// TIA Portal V19 export
FUNCTION "FC900_SafetyIntegration" : Void   // FC900, F_LAD
{ S7_Optimized_Access := 'TRUE' }
// stored: AutoNumber false
BEGIN

REGION Network 1: Bit de reset
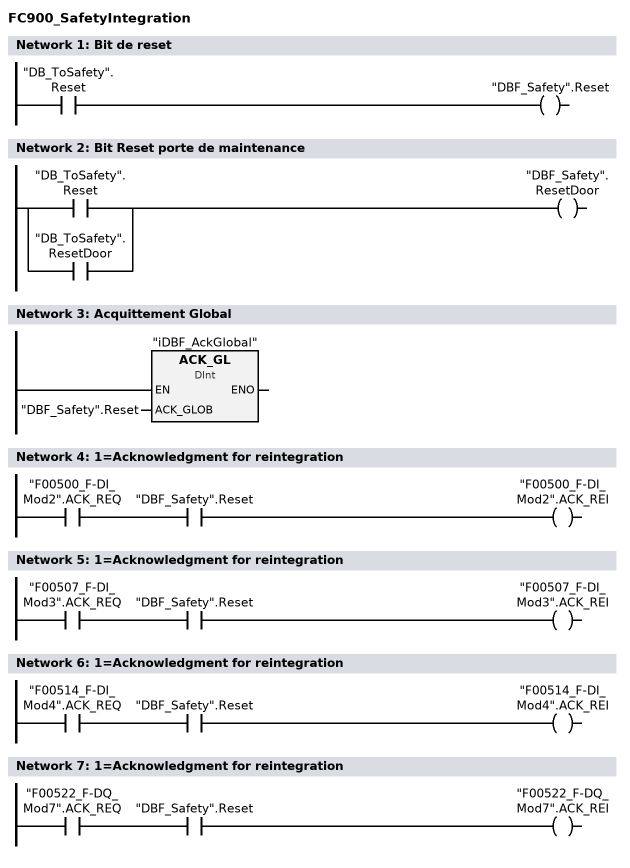
   RUNG wire#powerrail
      Contact( "DB_ToSafety".Reset )
      Coil( "DBF_Safety".Reset )
   END_RUNG
   // the same network as SCL:
   "DBF_Safety".Reset := "DB_ToSafety".Reset;
END_REGION

REGION Network 2: Bit Reset porte de maintenance
   RUNG wire#powerrail
      Contact( "DB_ToSafety".Reset )
      wire#w1
      Coil( "DBF_Safety".ResetDoor )
   END_RUNG
   RUNG wire#powerrail
      Contact( "DB_ToSafety".ResetDoor )
   END_RUNG wire#w1
   // the same network as SCL:
   "DBF_Safety".ResetDoor := "DB_ToSafety".Reset OR "DB_ToSafety".ResetDoor;
END_REGION

REGION Network 3: Acquittement Global
   RUNG wire#powerrail
      { S7_Templates := "codedbool_type := DInt" } "iDBF_AckGlobal".ACK_GL(ACK_GLOB := "DBF_Safety".Reset)
   END_RUNG
   // the same network as SCL:
   "iDBF_AckGlobal"(ACK_GLOB := "DBF_Safety".Reset);   // ACK_GL
END_REGION

REGION Network 4: 1=Acknowledgment for reintegration
   RUNG wire#powerrail
      Contact( "F00500_F-DI_Mod2".ACK_REQ )
      Contact( "DBF_Safety".Reset )
      Coil( "F00500_F-DI_Mod2".ACK_REI )
   END_RUNG
   // the same network as SCL:
   "F00500_F-DI_Mod2".ACK_REI := "F00500_F-DI_Mod2".ACK_REQ AND "DBF_Safety".Reset;
END_REGION

REGION Network 5: 1=Acknowledgment for reintegration
   RUNG wire#powerrail
      Contact( "F00507_F-DI_Mod3".ACK_REQ )
      Contact( "DBF_Safety".Reset )
      Coil( "F00507_F-DI_Mod3".ACK_REI )
   END_RUNG
   // the same network as SCL:
   "F00507_F-DI_Mod3".ACK_REI := "F00507_F-DI_Mod3".ACK_REQ AND "DBF_Safety".Reset;
END_REGION

REGION Network 6: 1=Acknowledgment for reintegration
   RUNG wire#powerrail
      Contact( "F00514_F-DI_Mod4".ACK_REQ )
      Contact( "DBF_Safety".Reset )
      Coil( "F00514_F-DI_Mod4".ACK_REI )
   END_RUNG
   // the same network as SCL:
   "F00514_F-DI_Mod4".ACK_REI := "F00514_F-DI_Mod4".ACK_REQ AND "DBF_Safety".Reset;
END_REGION

REGION Network 7: 1=Acknowledgment for reintegration
   RUNG wire#powerrail
      Contact( "F00522_F-DQ_Mod7".ACK_REQ )
      Contact( "DBF_Safety".Reset )
      Coil( "F00522_F-DQ_Mod7".ACK_REI )
   END_RUNG
   // the same network as SCL:
   "F00522_F-DQ_Mod7".ACK_REI := "F00522_F-DQ_Mod7".ACK_REQ AND "DBF_Safety".Reset;
END_REGION
END_FUNCTION
